INTERFACE I_Enumerable EXTENDS __SYSTEM.IQueryInterface

// Gets an enumerator that iterates through a collection. Returns TRUE if successful.
METHOD Get_Enumerator : BOOL;
VAR_INPUT
	ipEnumerator : REFERENCE TO I_Enumerator;
END_VAR
END_METHOD

END_INTERFACE

(* stored: Version 1.1.0.1, ProductVersion 3.1.4024.4
   Itf I_Enumerable: Id {d991723d-c59d-0fd8-04fd-3298c13d4437}
   Method Get_Enumerator: Id {7ac00d44-777f-070e-046d-7a145408ab43} *)
